FUNCTION_BLOCK SUBTRACTOR (* does y equals x1 minus x2 *)
  (* Standard: 61499-2 *)
  (* Version 11-01-12, GASR *)
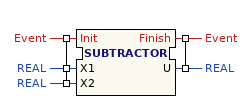
  EVENT_INPUT
    Init WITH X1, X2;
  END_EVENT
  EVENT_OUTPUT
    Finish WITH U;
  END_EVENT
  VAR_INPUT
    X1 : REAL;
    X2 : REAL;
  END_VAR
  VAR_OUTPUT
    U : REAL;
  END_VAR
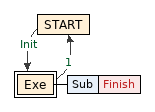
  EC_STATES
    Exe : Sub -> Finish;
    START;
  END_STATES
  EC_TRANSITIONS
    START TO Exe := Init;
    Exe TO START := 1;
  END_TRANSITIONS
  ALGORITHM Sub IN Lua:
U = X1 - X2
  END_ALGORITHM
END_FUNCTION_BLOCK
